FUNCTION_BLOCK TestActState2_HMI (* Service Interface Function Block Type *)
  (* Standard: 61499-2 *)
  (* Version 0.0, 6/3/2026, Schneider Electric, template *)
  PACKAGE SE.Nereda;
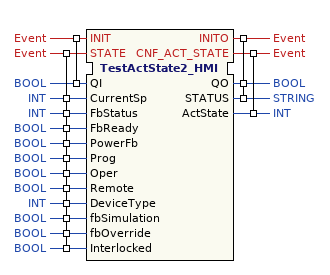
  EVENT_INPUT
    INIT WITH QI;
    STATE WITH CurrentSp, FbStatus, FbReady, PowerFb, Prog, Oper, Remote, DeviceType, fbSimulation, fbOverride, Interlocked;
  END_EVENT
  EVENT_OUTPUT
    INITO WITH QO, STATUS;
    CNF_ACT_STATE WITH ActState;
  END_EVENT
  VAR_INPUT
    QI : BOOL;
    CurrentSp : INT;
    FbStatus : INT;
    FbReady : BOOL;
    PowerFb : BOOL;
    Prog : BOOL;
    Oper : BOOL;
    Remote : BOOL;
    DeviceType : INT;
    fbSimulation : BOOL;
    fbOverride : BOOL;
    Interlocked : BOOL;
  END_VAR
  VAR_OUTPUT
    QO : BOOL; (* Event Output Qualifier *)
    STATUS : STRING; (* Service Status *)
    ActState : INT;
  END_VAR
  SERVICE /
    SEQUENCE 
    END_SEQUENCE
  END_SERVICE
END_FUNCTION_BLOCK
